// TIA Portal V18 export
// export: Created 2026-06-08T16:52:57.1419064Z, ExportSetting WithDefaults, DisplayName Totally Integrated Automation Portal, DisplayVersion V18, DisplayName TIA Portal Openness, DisplayVersion V18, DisplayName TIA Portal Version Control Interface, DisplayVersion V18, DisplayName STEP 7 Professional, DisplayVersion V18, DisplayName STEP 7 Safety, DisplayVersion V18, DisplayName WinCC Professional, DisplayVersion V18
ORGANIZATION_BLOCK "Cyclic interrupt"   // OB30, LAD, CyclicInterrupt
{ S7_Optimized_Access := 'TRUE' }
VERSION : 0.1
// stored: AutoNumber true, IsIECCheckEnabled false, SetENOAutomatically false
   VAR_INPUT
      Initial_Call : Bool;   // Initial call of this OB
      Event_Count : Int;   // Events discarded
   END_VAR
BEGIN

REGION Network 1
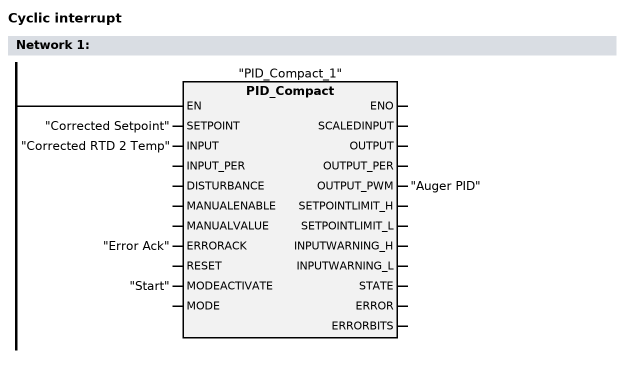
   RUNG wire#powerrail
      "PID_Compact_1".PID_Compact(Setpoint := "Corrected Setpoint", Input := "Corrected RTD 2 Temp", Input_PER :=, Disturbance :=, ManualEnable :=, ManualValue :=, ErrorAck := "Error Ack", Reset :=, ModeActivate := "Start", Mode :=, ScaledInput =>, Output =>, Output_PER =>, Output_PWM => "Auger PID", SetpointLimit_H =>, SetpointLimit_L =>, InputWarning_H =>, InputWarning_L =>, State =>, Error =>, ErrorBits =>)
   END_RUNG
   // the same network as SCL:
   "PID_Compact_1"(Setpoint := "Corrected Setpoint",   // PID_Compact
                   Input := "Corrected RTD 2 Temp",
                   ErrorAck := "Error Ack",
                   ModeActivate := "Start",
                   Output_PWM => "Auger PID");
END_REGION
END_ORGANIZATION_BLOCK
